FUNCTION CheckDivReal  : REAL
VAR_INPUT
	divisor : REAL;
END_VAR
VAR
END_VAR

IF divisor = 0 THEN
        CheckDivReal := 1E-10;
ELSE
        CheckDivReal := divisor;
END_IF

END_FUNCTION

(* stored: Version 1.1.0.1, ProductVersion 3.1.4022.18
   POU CheckDivReal: Id {d9169663-c48d-4095-a4da-7d280d972d6e}, SpecialFunc None *)
